TYPE HEATType :
(
	HEATType_Default := 0, // 常规的加热,两者都具备
	HEATType_Smart := 1, // 智能加热
	HEATType_Manul := 2 // 手动加热
)UINT;
END_TYPE

(* stored: Version 1.1.0.1, ProductVersion 3.1.4024.4
   DUT HEATType: Id {11e0770f-475c-464f-87e8-4a80555adb09} *)
